Staubli VAL3: encSetDrvPwrAck.pgx

public program encSetDrvPwrAck()
begin
  // Copyright (c) 2021, Institute for Factory Automation and Production Systems (FAPS)
  //
  // Licensed under the Apache License, Version 2.0 (the "License");
  // you may not use this file except in compliance with the License.
  // You may obtain a copy of the License at
  //
  //     http://www.apache.org/licenses/LICENSE-2.0
  //
  // Unless required by applicable law or agreed to in writing, software
  // distributed under the License is distributed on an "AS IS" BASIS,
  // WITHOUT WARRANTIES OR CONDITIONS OF ANY KIND, either express or implied.
  // See the License for the specific language governing permissions and
  // limitations under the License.


  // encode 'prefix' and 'header'
  call SimpleMsg:encPrefixHeader(setDrvPwrAck.prefix,setDrvPwrAck.header)

  // encodings of the body field (dummy data) is ignored to save CPU time, since values are all zeros
end
